// TIA Portal V18 export
FUNCTION "Servo" : Void   // FC2500, LAD
{ S7_Optimized_Access := 'TRUE' }
// stored: AutoNumber false, SetENOAutomatically false
BEGIN

REGION Network 1
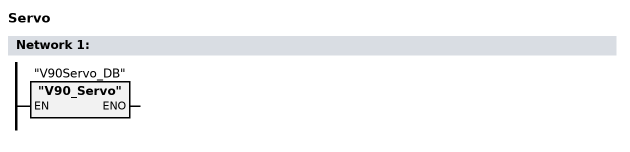
   RUNG wire#powerrail
      "V90Servo_DB"()
   END_RUNG
   // the same network as SCL:
   "V90Servo_DB"();   // "V90_Servo"
END_REGION
END_FUNCTION
